(* IEC 61131-3 sources: SmartHomeNew/snapshots/project_clean_state_2026_04_16/workspace/dut_rebuild/blinds_v2/extraction, 1 file *)

(* ---- FB_Blinds_Command_Extractor_DRAFT.st ---- *)
FUNCTION_BLOCK FB_Blinds_Command_Extractor_DRAFT
VAR_INPUT
    VI_Position_Setpoint : BYTE;
    VI_Manual_Override : BOOL;
END_VAR
VAR_OUTPUT
    VO_Command : ST_Blinds_Command_V2;
END_VAR

VO_Command.Position_Setpoint := VI_Position_Setpoint;
VO_Command.Manual_Override := VI_Manual_Override;
END_FUNCTION_BLOCK
